(* PLC project conveyor_v2.project, CODESYS CODESYS V3.5 SP22 Patch 3 *)
(* stored: creationDateTime 2026-09-17T15:43:22.0964234, modificationDateTime 2026-09-17T15:39:54.6608792 *)

PROGRAM PLC_PRG
  VAR
    bStart AT %IX0.0 : BOOL;  (* Nút Start (NO) *)
    bStop AT %IX0.1 : BOOL;  (* Nút Stop (NC) *)
    bSensorIn AT %IX0.2 : BOOL;  (* Cảm biến sản phẩm *)
    bReset AT %IX0.3 : BOOL;  (* Nút reset bộ đếm *)
    bEStop AT %IX0.4 : BOOL;  (* Dừng khẩn (NC) *)
    bMotor AT %QX0.0 : BOOL;  (* Contactor băng tải *)
    bLampDone AT %QX0.3 : BOOL;  (* Đèn báo đủ số lượng *)
  END_VAR
  VAR
    fbCounter : CTU;  (* Bộ đếm sản phẩm *)
    iCount : INT;
    iPreset : INT := 20;
  END_VAR

                    fbCounter(CU := bSensorIn AND bMotor, RESET := bReset, PV := iPreset,
          Q => bLampDone, CV => iCount);

bMotor := (bStart OR bMotor) AND bStop AND bEStop AND NOT bLampDone;
                  
END_PROGRAM

CONFIGURATION Device
  RESOURCE Application ON PLC
    TASK MainTask(INTERVAL := T#20ms, PRIORITY := 1);
    PROGRAM PLC_PRG WITH MainTask : PLC_PRG;
  END_RESOURCE
END_CONFIGURATION
